PROGRAM p_StatusLights
VAR
END_VAR

gxRedLight := xEnableRemoteControl;//Remote control in use
gxGreenLight := NOT (gxRedLight OR gxYellowLight); (* attach system error or something here someday *)

END_PROGRAM

(* stored: Version 1.1.0.1, ProductVersion 3.1.4022.18
   POU p_StatusLights: Id {614a6145-0e85-4695-9427-e36cd2542668}, SpecialFunc None *)
